{attribute 'linkalways'} 
{attribute 'no_explicit_call' := 'This FB is a CLASS and must be accessed using methods or properties'}
{attribute 'enable_dynamic_creation'}
FUNCTION_BLOCK _ETcVnLayerNameType EXTENDS EnumDatatypeBase
VAR
	localData : ETcVnLayerNameType;
	activeData : REFERENCE TO ETcVnLayerNameType;
	enumBaseDatatype : _DINT(localData);
END_VAR

METHOD PRIVATE AddLocalEnumeration
VAR_INPUT
	Enumeration : T_MAXSTRING;
	Value : ETcVnLayerNameType;
END_VAR
AddEnumeration(Enumeration, Value);
END_METHOD

PROPERTY PUBLIC Address : PVOID
GET
Address := ADR(activeData);
END_GET
END_PROPERTY

METHOD PUBLIC ClearReference
VAR_INPUT
END_VAR
activeData REF= localData;
SetBaseDatatypeReference();
END_METHOD

METHOD PUBLIC Clone : I_Datatype
VAR
    pClone : POINTER TO _ETcVnLayerNameType;
END_VAR
pClone := __NEW(_ETcVnLayerNameType(InitialValue := Value));
Clone := pClone^;
END_METHOD

METHOD FB_init : BOOL
VAR_INPUT
	bInitRetains : BOOL; // if TRUE, the retain variables are initialized (warm start / cold start)
	bInCopyCode : BOOL;  // if TRUE, the instance afterwards gets moved into the copy code (online change)
	InitialValue : ETcVnLayerNameType;
END_VAR
localData := InitialValue;
AddBaseDatatype(enumBaseDatatype);
ClearReference();

AddLocalEnumeration('TCVN_LNT_ALL', ETcVnLayerNameType.TCVN_LNT_ALL);
AddLocalEnumeration('TCVN_LNT_OUTPUTS', ETcVnLayerNameType.TCVN_LNT_OUTPUTS);
AddLocalEnumeration('TCVN_LNT_INPUTS', ETcVnLayerNameType.TCVN_LNT_INPUTS);
END_METHOD

PROPERTY PUBLIC Identifier : T_MAXSTRING
GET
Identifier := 'ETcVnLayerNameType';
END_GET
END_PROPERTY

METHOD IsEnumeratorValueEqual : BOOL
VAR_INPUT
	Enumerator : I_KeyValueForwardEnumerator;
END_VAR
VAR
	storedValue : ETcVnLayerNameType;
END_VAR
IF NOT Enumerator.TryGet(storedValue) THEN
	RETURN;
END_IF

IsEnumeratorValueEqual := storedValue = activeData;
END_METHOD

METHOD PUBLIC MakeReferenceTo
VAR_INPUT
	ReferenceTarget : REFERENCE TO ETcVnLayerNameType;
END_VAR
activeData REF= ReferenceTarget;
SetBaseDatatypeReference();
END_METHOD

METHOD PROTECTED SetBaseDatatypeReference
VAR_INPUT
END_VAR
enumBaseDatatype.MakeReferenceTo(activeData);
END_METHOD

PROPERTY PUBLIC Size : UDINT
GET
Size := SIZEOF(activeData);
END_GET
END_PROPERTY

METHOD TryMakeReferenceTo : BOOL
VAR_INPUT
	Target : I_Datatype;
END_VAR
VAR
	pTargetData : POINTER TO ETcVnLayerNameType;
END_VAR
IF NOT IsEquivalentTo(Target) THEN
	RETURN;
END_IF

pTargetData := Target.Address;
activeData REF= pTargetData^;
SetBaseDatatypeReference();
TryMakeReferenceTo := TRUE;
END_METHOD

PROPERTY PUBLIC Value : ETcVnLayerNameType
GET
Value := activeData;
END_GET
SET
activeData := Value;
END_SET
END_PROPERTY

END_FUNCTION_BLOCK

(* stored: Version 1.1.0.1, ProductVersion 3.1.4024.15
   POU _ETcVnLayerNameType: Id {5e2c1f45-536c-0b62-36d9-024f18dafd29}, SpecialFunc None
   Folder Core: Id {a349abfa-9ff0-053d-24f3-d2b8722db3c4}
   Folder Protected: Id {e0a92cf6-4d61-0a65-1c68-1b37ed7630b9}
   Folder Customize: Id {a9a83900-770e-046d-1126-c9addf6e6f68}
   Folder Constructor: Id {fe3be51d-16b1-088a-0bda-ed9d2b757956}
   Folder Private: Id {96a1f913-cb33-0028-3e11-f142653f7163}
   Folder Protected: Id {dfba0cad-6610-0af3-3888-1ff66d8ee017}
   Method AddLocalEnumeration: Id {f167b1f5-3118-024b-29fc-2da53551f646}
   Property Address: Id {c2f5289a-231f-054e-2a60-ae2448ca33e3}
   Get Get: Id {1dcbe5d2-c89e-062b-360d-4882732c3366}
   Method ClearReference: Id {21706834-62e3-09ad-17f5-3b3f3fb5d5d2}
   Method Clone: Id {2ecf9df0-5282-0daf-1e6c-136fab984e85}
   Method FB_init: Id {d331963e-82ac-0bbc-0350-62fd167d5363}
   Property Identifier: Id {f1faad00-07ae-04e4-084f-91f82227ac04}
   Get Get: Id {efe4e335-73dd-0e3b-3657-ea3824b51976}
   Method IsEnumeratorValueEqual: Id {d71b3300-5386-0d9d-2f6d-6230fcce5216}
   Method MakeReferenceTo: Id {0804218c-b8a7-09e5-1151-7e6706b38a0f}
   Method SetBaseDatatypeReference: Id {59cb214e-2a32-0bb0-30f9-c0668024f4c6}
   Property Size: Id {3a519f40-e583-0263-3b61-92cc32ee2982}
   Get Get: Id {435082ff-10a8-09ea-1cd5-e7493f006df2}
   Method TryMakeReferenceTo: Id {a7460f70-8074-0072-11c7-79d5fcfc246d}
   Property Value: Id {3f9836b5-4512-0660-1e0a-592b7439c0f7}
   Get Get: Id {87426358-dabe-0603-01ea-4af2a6e9c6f0}
   Set Set: Id {74158932-5f14-046c-2a72-76b5b2b56467} *)
